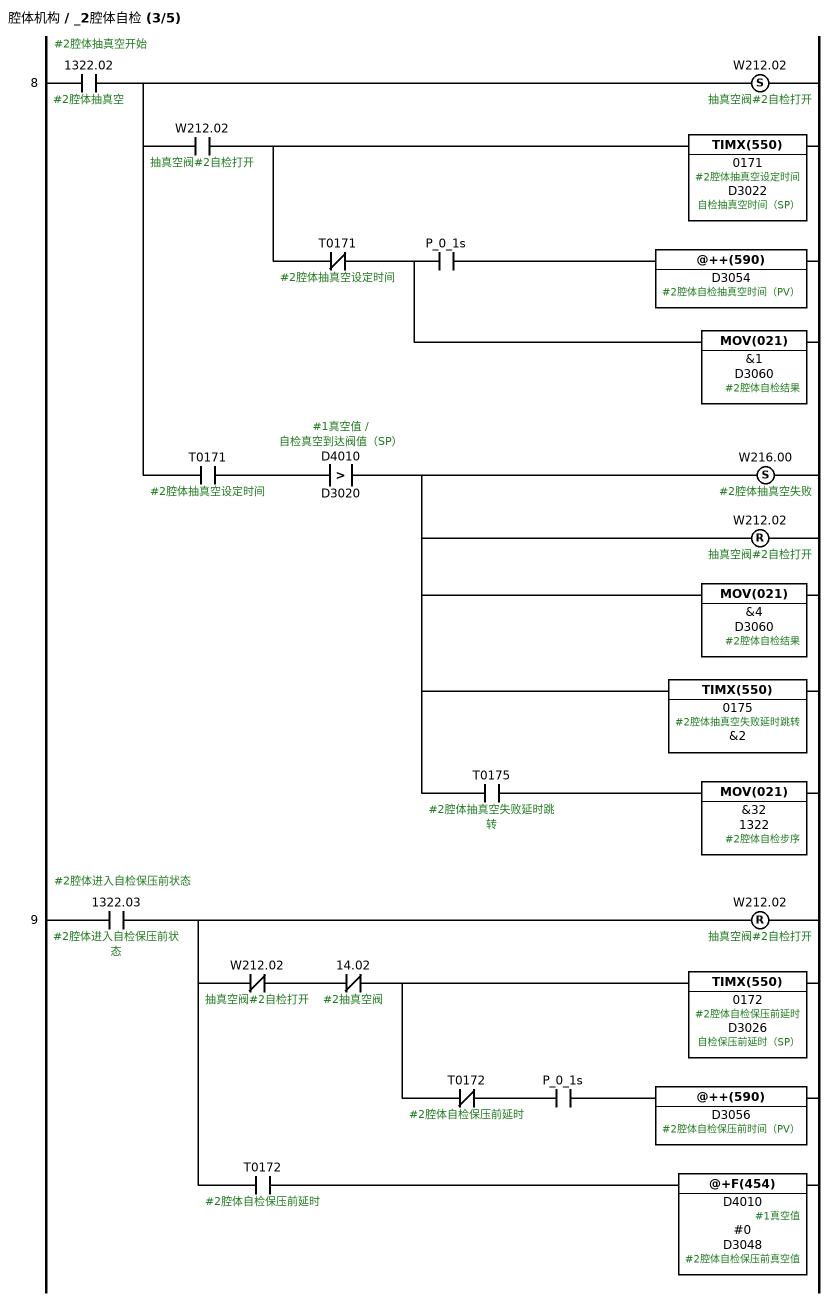
; [picture p312: 腔体机构 / _2腔体自检, rungs 8-9]
; rung 8: #2腔体抽真空开始
LD 1322.02  ; #2腔体抽真空
OUT TR0
SET W212.02  ; 抽真空阀#2自检打开
AND W212.02  ; 抽真空阀#2自检打开
TIMX(550) 0171 D3022  ; 自检抽真空时间（SP）, #2腔体抽真空设定时间
ANDNOT T0171  ; #2腔体抽真空设定时间
OUT TR1
AND P_0_1s
@++(590) D3054  ; #2腔体自检抽真空时间（PV）
LD TR1
MOV(021) &1 D3060  ; #2腔体自检结果
LD TR0
AND T0171  ; #2腔体抽真空设定时间
AND>F(333) D4010 D3020  ; #1真空值, 自检真空到达阀值（SP）
SET W216.00  ; #2腔体抽真空失败
RSET W212.02  ; 抽真空阀#2自检打开
MOV(021) &4 D3060  ; #2腔体自检结果
TIMX(550) 0175 &2  ; #2腔体抽真空失败延时跳转
AND T0175  ; #2腔体抽真空失败延时跳转
MOV(021) &32 1322  ; #2腔体自检步序
; rung 9: #2腔体进入自检保压前状态
LD 1322.03  ; #2腔体进入自检保压前状态
OUT TR0
RSET W212.02  ; 抽真空阀#2自检打开
ANDNOT W212.02  ; 抽真空阀#2自检打开
ANDNOT 14.02  ; #2抽真空阀
TIMX(550) 0172 D3026  ; 自检保压前延时（SP）, #2腔体自检保压前延时
ANDNOT T0172  ; #2腔体自检保压前延时
AND P_0_1s
@++(590) D3056  ; #2腔体自检保压前时间（PV）
LD TR0
AND T0172  ; #2腔体自检保压前延时
@+F(454) D4010 #0 D3048  ; #1真空值, #2腔体自检保压前真空值

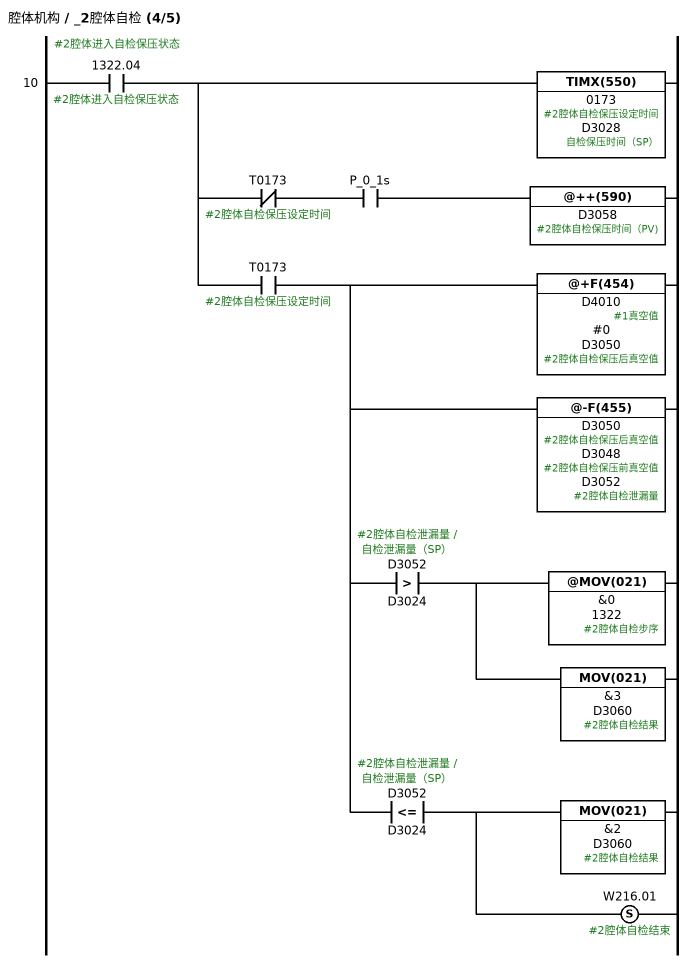
; rung 10: #2腔体进入自检保压状态
LD 1322.04  ; #2腔体进入自检保压状态
OUT TR0
TIMX(550) 0173 D3028  ; 自检保压时间（SP）, #2腔体自检保压设定时间
ANDNOT T0173  ; #2腔体自检保压设定时间
AND P_0_1s
@++(590) D3058  ; #2腔体自检保压时间（PV)
LD TR0
AND T0173  ; #2腔体自检保压设定时间
OUT TR0
@+F(454) D4010 #0 D3050  ; #1真空值, #2腔体自检保压后真空值
@-F(455) D3050 D3048 D3052  ; #2腔体自检保压后真空值, #2腔体自检保压前真空值, #2腔体自检泄漏量
AND>F(333) D3052 D3024  ; #2腔体自检泄漏量, 自检泄漏量（SP）
@MOV(021) &0 1322  ; #2腔体自检步序
MOV(021) &3 D3060  ; #2腔体自检结果
LD TR0
AND<=F(332) D3052 D3024  ; #2腔体自检泄漏量, 自检泄漏量（SP）
MOV(021) &2 D3060  ; #2腔体自检结果
SET W216.01  ; #2腔体自检结束

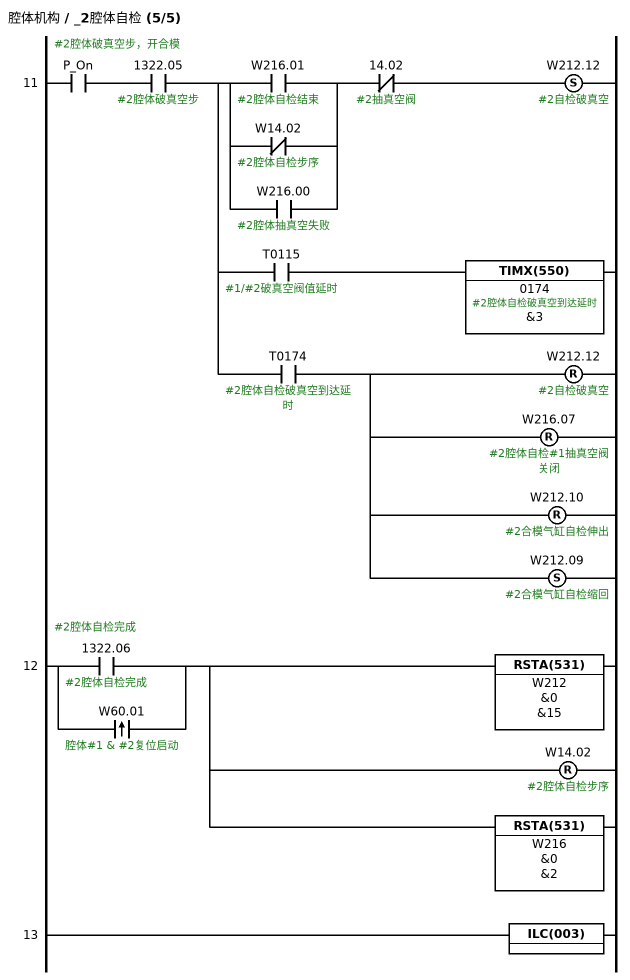
; rung 11: #2腔体破真空步，开合模
LD P_On
AND 1322.05  ; #2腔体破真空步
OUT TR0
LD W216.01  ; #2腔体自检结束
ORNOT W14.02  ; #2腔体自检步序
OR W216.00  ; #2腔体抽真空失败
ANDLD
ANDNOT 14.02  ; #2抽真空阀
SET W212.12  ; #2自检破真空
LD TR0
AND T0115  ; #1/#2破真空阀值延时
TIMX(550) 0174 &3  ; #2腔体自检破真空到达延时
LD TR0
AND T0174  ; #2腔体自检破真空到达延时
RSET W212.12  ; #2自检破真空
RSET W216.07  ; #2腔体自检#1抽真空阀关闭
RSET W212.10  ; #2合模气缸自检伸出
SET W212.09  ; #2合模气缸自检缩回
; rung 12: #2腔体自检完成
LD 1322.06  ; #2腔体自检完成
@OR W60.01  ; 腔体#1 & #2复位启动
RSTA(531) W212 &0 &15
RSET W14.02  ; #2腔体自检步序
RSTA(531) W216 &0 &2
; rung 13
ILC(003)

### Section _3腔体自检

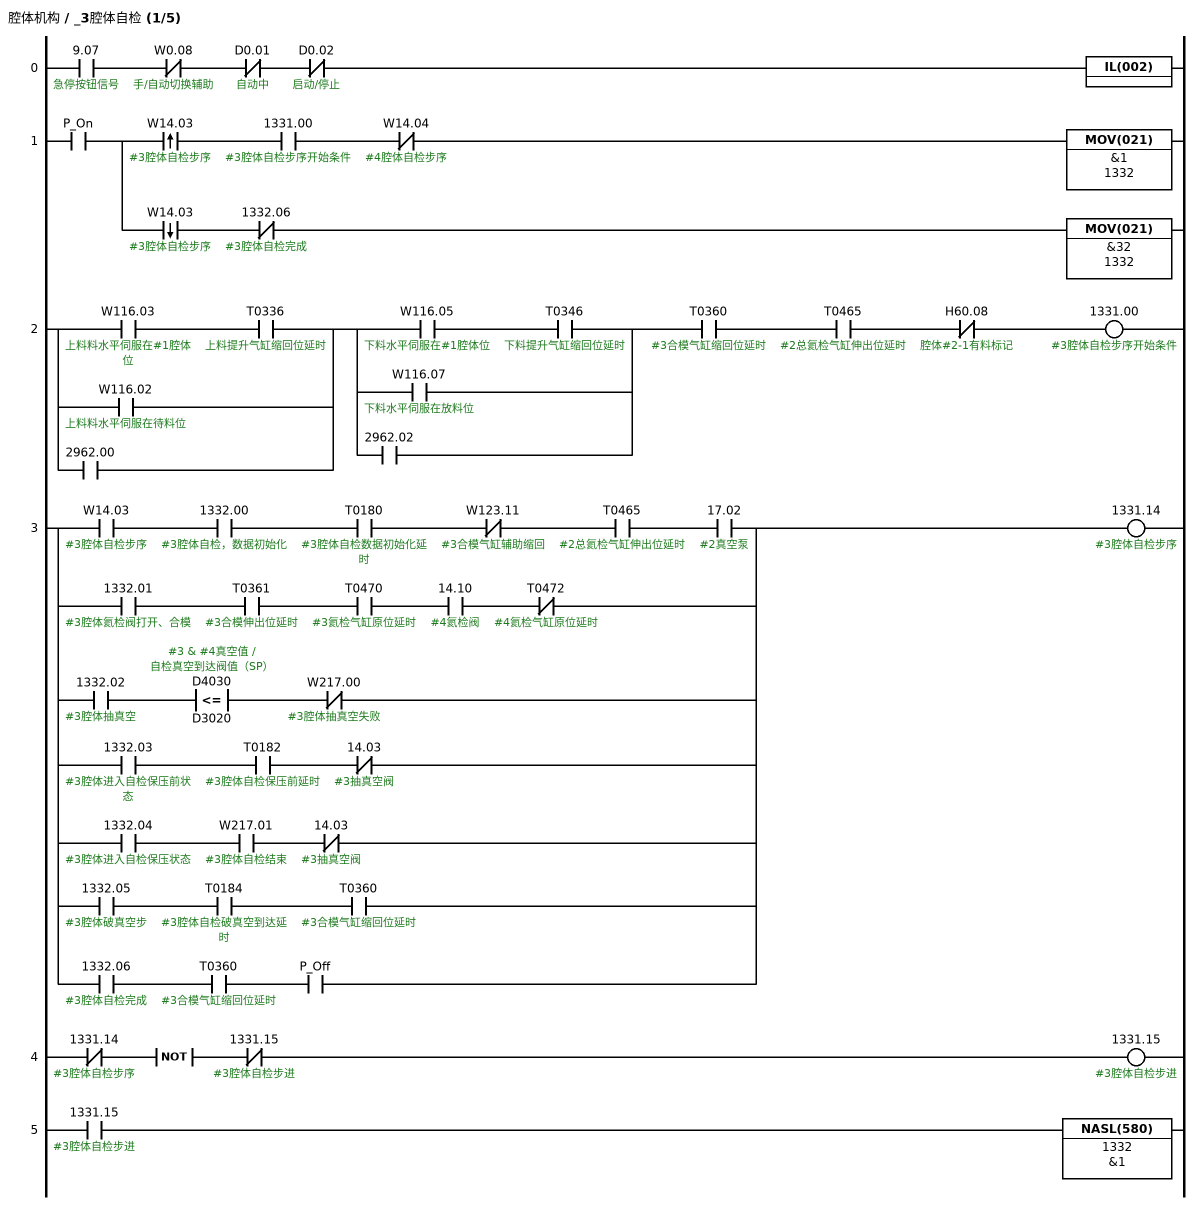
; rung 0
LD 9.07  ; 急停按钮信号
ANDNOT W0.08  ; 手/自动切换辅助
ANDNOT D0.01  ; 自动中
ANDNOT D0.02  ; 启动/停止
IL(002)
; rung 1
LD P_On
OUT TR0
@AND W14.03  ; #3腔体自检步序
AND 1331.00  ; #3腔体自检步序开始条件
ANDNOT W14.04  ; #4腔体自检步序
MOV(021) &1 1332
LD TR0
%AND W14.03  ; #3腔体自检步序
ANDNOT 1332.06  ; #3腔体自检完成
MOV(021) &32 1332
; rung 2
LD W116.03  ; 上料料水平伺服在#1腔体位
AND T0336  ; 上料提升气缸缩回位延时
OR W116.02  ; 上料料水平伺服在待料位
OR 2962.00
LD W116.05  ; 下料水平伺服在#1腔体位
AND T0346  ; 下料提升气缸缩回位延时
OR W116.07  ; 下料水平伺服在放料位
OR 2962.02
ANDLD
AND T0360  ; #3合模气缸缩回位延时
AND T0465  ; #2总氦检气缸伸出位延时
ANDNOT H60.08  ; 腔体#2-1有料标记
OUT 1331.00  ; #3腔体自检步序开始条件
; rung 3
LD W14.03  ; #3腔体自检步序
AND 1332.00  ; #3腔体自检，数据初始化
AND T0180  ; #3腔体自检数据初始化延时
ANDNOT W123.11  ; #3合模气缸辅助缩回
AND T0465  ; #2总氦检气缸伸出位延时
AND 17.02  ; #2真空泵
LD 1332.01  ; #3腔体氦检阀打开、合模
AND T0361  ; #3合模伸出位延时
AND T0470  ; #3氦检气缸原位延时
AND 14.10  ; #4氦检阀
ANDNOT T0472  ; #4氦检气缸原位延时
ORLD
LD 1332.02  ; #3腔体抽真空
AND<=F(332) D4030 D3020  ; #3 & #4真空值, 自检真空到达阀值（SP）
ANDNOT W217.00  ; #3腔体抽真空失败
ORLD
LD 1332.03  ; #3腔体进入自检保压前状态
AND T0182  ; #3腔体自检保压前延时
ANDNOT 14.03  ; #3抽真空阀
ORLD
LD 1332.04  ; #3腔体进入自检保压状态
AND W217.01  ; #3腔体自检结束
ANDNOT 14.03  ; #3抽真空阀
ORLD
LD 1332.05  ; #3腔体破真空步
AND T0184  ; #3腔体自检破真空到达延时
AND T0360  ; #3合模气缸缩回位延时
ORLD
LD 1332.06  ; #3腔体自检完成
AND T0360  ; #3合模气缸缩回位延时
AND P_Off
ORLD
OUT 1331.14  ; #3腔体自检步序
; rung 4
LDNOT 1331.14  ; #3腔体自检步序
NOT(520)
ANDNOT 1331.15  ; #3腔体自检步进
OUT 1331.15  ; #3腔体自检步进
; rung 5
LD 1331.15  ; #3腔体自检步进
NASL(580) 1332 &1

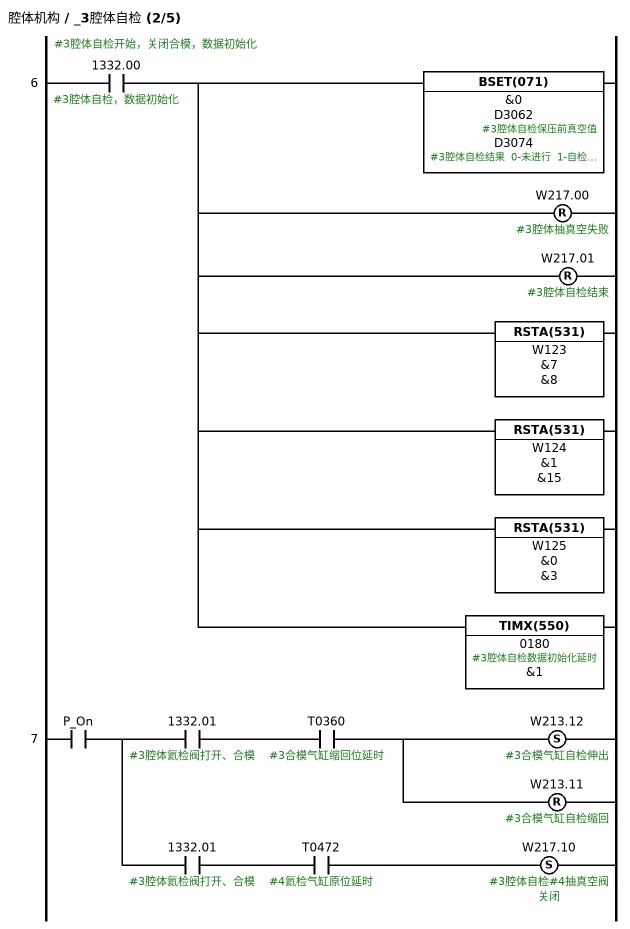
; rung 6: #3腔体自检开始，关闭合模，数据初始化
LD 1332.00  ; #3腔体自检，数据初始化
BSET(071) &0 D3062 D3074  ; #3腔体自检保压前真空值, #3腔体自检结果  0-未进行  1-自检中  2-自检OK  3-自检泄漏  4-自检抽真空NG
RSET W217.00  ; #3腔体抽真空失败
RSET W217.01  ; #3腔体自检结束
RSTA(531) W123 &7 &8
RSTA(531) W124 &1 &15
RSTA(531) W125 &0 &3
TIMX(550) 0180 &1  ; #3腔体自检数据初始化延时
; rung 7
LD P_On
OUT TR0
AND 1332.01  ; #3腔体氦检阀打开、合模
AND T0360  ; #3合模气缸缩回位延时
SET W213.12  ; #3合模气缸自检伸出
RSET W213.11  ; #3合模气缸自检缩回
LD TR0
AND 1332.01  ; #3腔体氦检阀打开、合模
AND T0472  ; #4氦检气缸原位延时
SET W217.10  ; #3腔体自检#4抽真空阀关闭

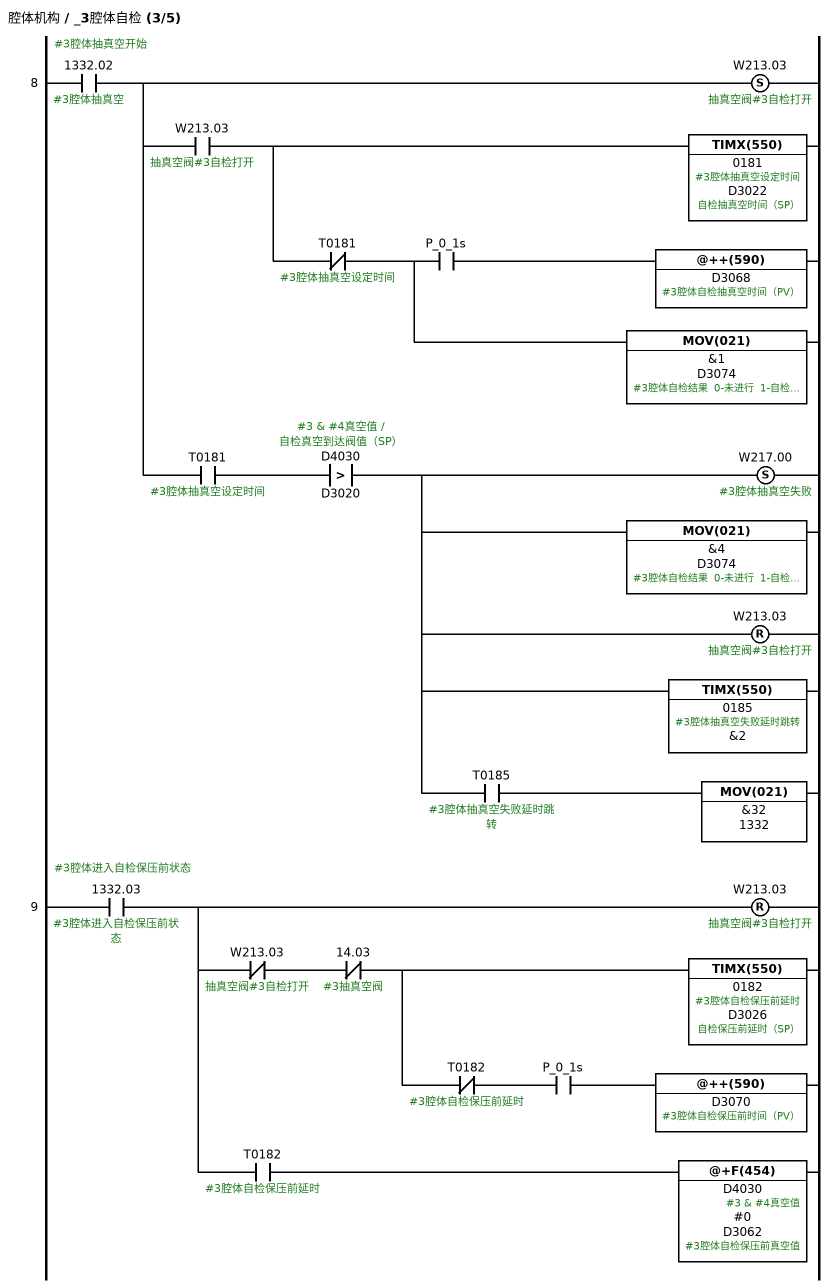
; rung 8: #3腔体抽真空开始
LD 1332.02  ; #3腔体抽真空
OUT TR0
SET W213.03  ; 抽真空阀#3自检打开
AND W213.03  ; 抽真空阀#3自检打开
TIMX(550) 0181 D3022  ; 自检抽真空时间（SP）, #3腔体抽真空设定时间
ANDNOT T0181  ; #3腔体抽真空设定时间
OUT TR1
AND P_0_1s
@++(590) D3068  ; #3腔体自检抽真空时间（PV）
LD TR1
MOV(021) &1 D3074  ; #3腔体自检结果  0-未进行  1-自检中  2-自检OK  3-自检泄漏  4-自检抽真空NG
LD TR0
AND T0181  ; #3腔体抽真空设定时间
AND>F(333) D4030 D3020  ; #3 & #4真空值, 自检真空到达阀值（SP）
SET W217.00  ; #3腔体抽真空失败
MOV(021) &4 D3074  ; #3腔体自检结果  0-未进行  1-自检中  2-自检OK  3-自检泄漏  4-自检抽真空NG
RSET W213.03  ; 抽真空阀#3自检打开
TIMX(550) 0185 &2  ; #3腔体抽真空失败延时跳转
AND T0185  ; #3腔体抽真空失败延时跳转
MOV(021) &32 1332
; rung 9: #3腔体进入自检保压前状态
LD 1332.03  ; #3腔体进入自检保压前状态
OUT TR0
RSET W213.03  ; 抽真空阀#3自检打开
ANDNOT W213.03  ; 抽真空阀#3自检打开
ANDNOT 14.03  ; #3抽真空阀
TIMX(550) 0182 D3026  ; 自检保压前延时（SP）, #3腔体自检保压前延时
ANDNOT T0182  ; #3腔体自检保压前延时
AND P_0_1s
@++(590) D3070  ; #3腔体自检保压前时间（PV）
LD TR0
AND T0182  ; #3腔体自检保压前延时
@+F(454) D4030 #0 D3062  ; #3 & #4真空值, #3腔体自检保压前真空值

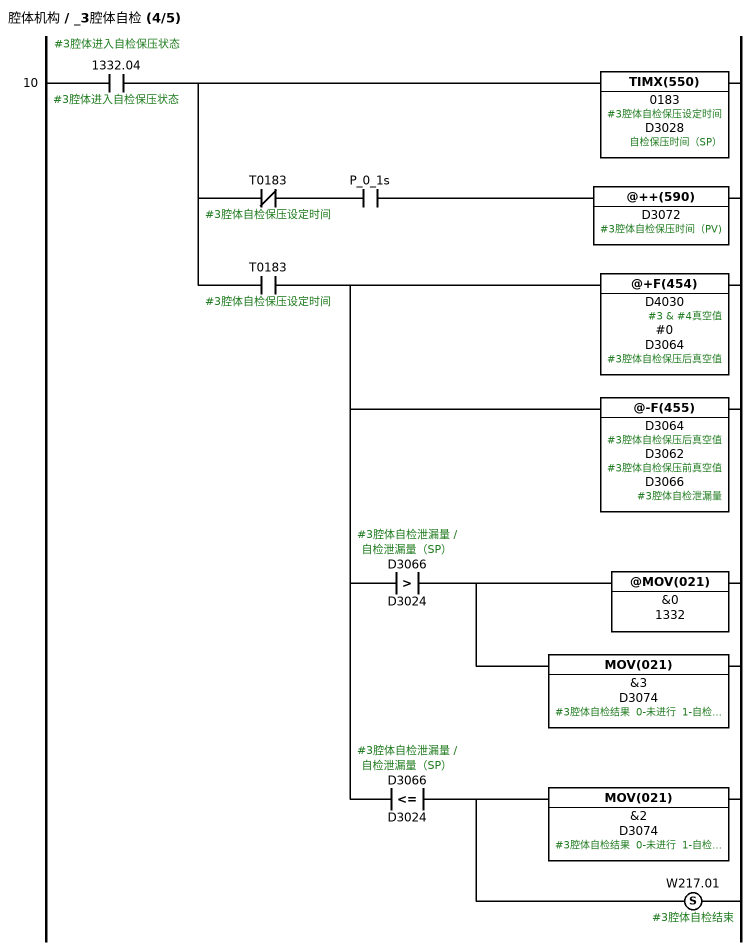
; rung 10: #3腔体进入自检保压状态
LD 1332.04  ; #3腔体进入自检保压状态
OUT TR0
TIMX(550) 0183 D3028  ; 自检保压时间（SP）, #3腔体自检保压设定时间
ANDNOT T0183  ; #3腔体自检保压设定时间
AND P_0_1s
@++(590) D3072  ; #3腔体自检保压时间（PV)
LD TR0
AND T0183  ; #3腔体自检保压设定时间
OUT TR0
@+F(454) D4030 #0 D3064  ; #3 & #4真空值, #3腔体自检保压后真空值
@-F(455) D3064 D3062 D3066  ; #3腔体自检保压后真空值, #3腔体自检保压前真空值, #3腔体自检泄漏量
AND>F(333) D3066 D3024  ; #3腔体自检泄漏量, 自检泄漏量（SP）
@MOV(021) &0 1332
MOV(021) &3 D3074  ; #3腔体自检结果  0-未进行  1-自检中  2-自检OK  3-自检泄漏  4-自检抽真空NG
LD TR0
AND<=F(332) D3066 D3024  ; #3腔体自检泄漏量, 自检泄漏量（SP）
MOV(021) &2 D3074  ; #3腔体自检结果  0-未进行  1-自检中  2-自检OK  3-自检泄漏  4-自检抽真空NG
SET W217.01  ; #3腔体自检结束

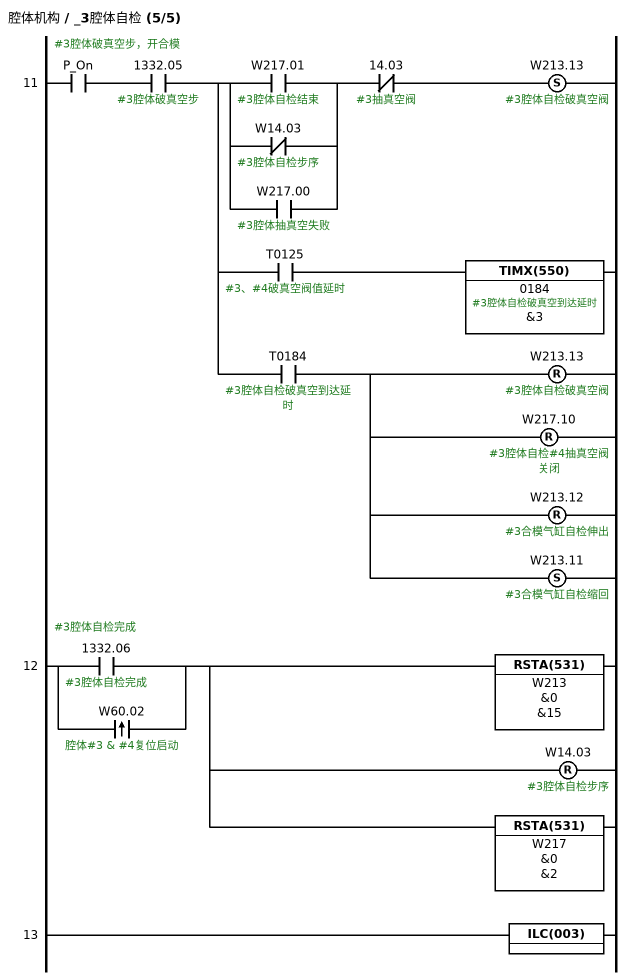
; rung 11: #3腔体破真空步，开合模
LD P_On
AND 1332.05  ; #3腔体破真空步
OUT TR0
LD W217.01  ; #3腔体自检结束
ORNOT W14.03  ; #3腔体自检步序
OR W217.00  ; #3腔体抽真空失败
ANDLD
ANDNOT 14.03  ; #3抽真空阀
SET W213.13  ; #3腔体自检破真空阀
LD TR0
AND T0125  ; #3、#4破真空阀值延时
TIMX(550) 0184 &3  ; #3腔体自检破真空到达延时
LD TR0
AND T0184  ; #3腔体自检破真空到达延时
RSET W213.13  ; #3腔体自检破真空阀
RSET W217.10  ; #3腔体自检#4抽真空阀关闭
RSET W213.12  ; #3合模气缸自检伸出
SET W213.11  ; #3合模气缸自检缩回
; rung 12: #3腔体自检完成
LD 1332.06  ; #3腔体自检完成
@OR W60.02  ; 腔体#3 & #4复位启动
RSTA(531) W213 &0 &15
RSET W14.03  ; #3腔体自检步序
RSTA(531) W217 &0 &2
; rung 13
ILC(003)

### Section _4腔体自检

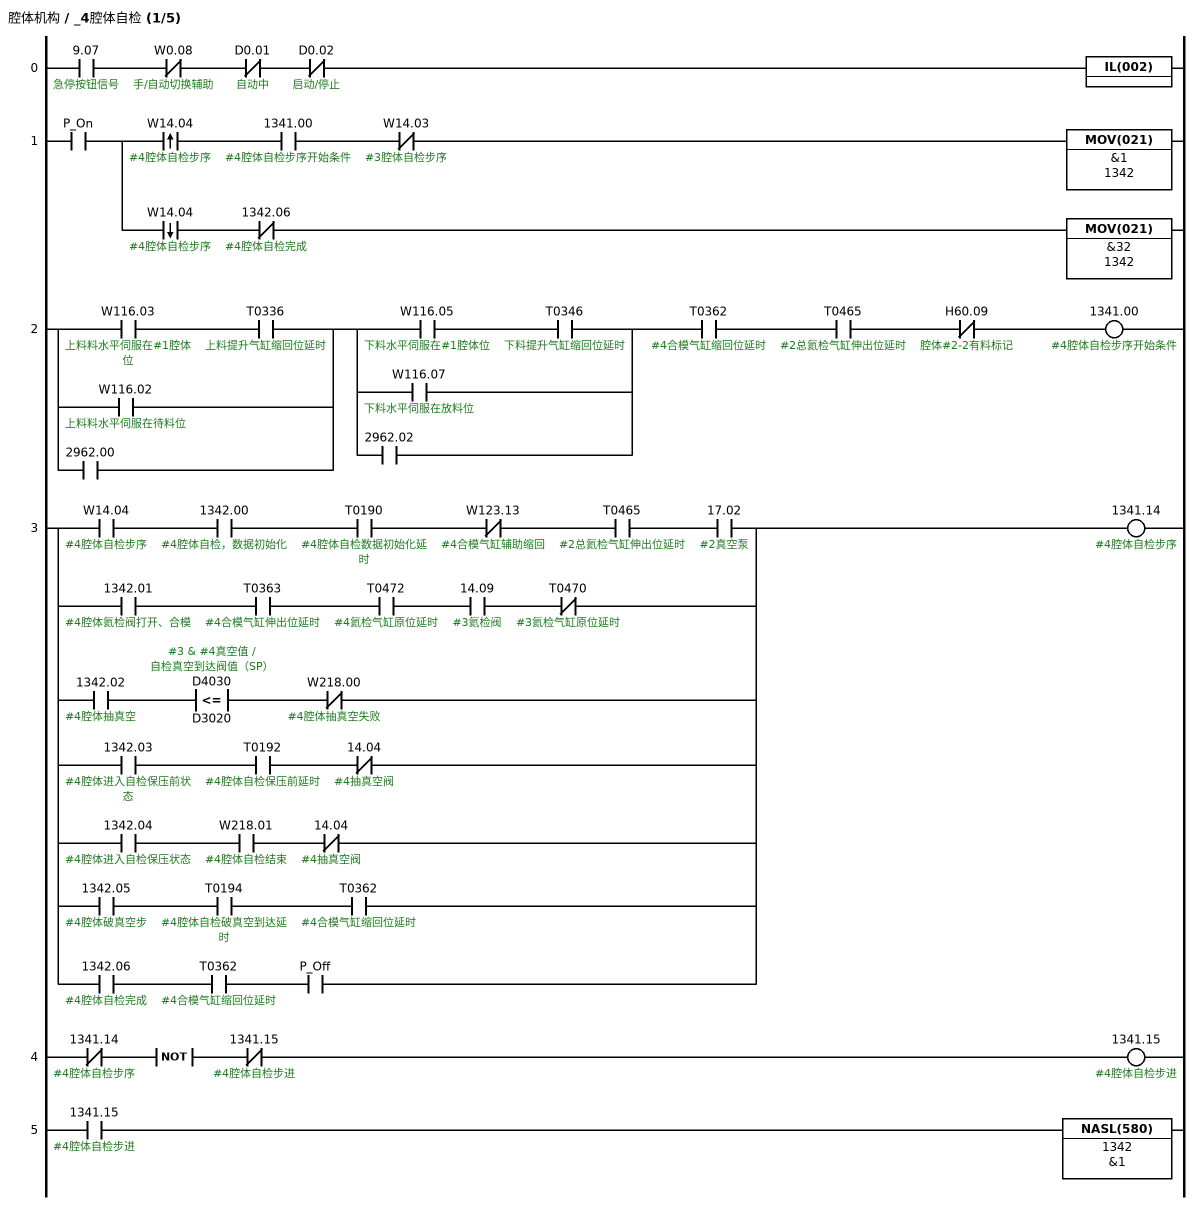
; rung 0
LD 9.07  ; 急停按钮信号
ANDNOT W0.08  ; 手/自动切换辅助
ANDNOT D0.01  ; 自动中
ANDNOT D0.02  ; 启动/停止
IL(002)
; rung 1
LD P_On
OUT TR0
@AND W14.04  ; #4腔体自检步序
AND 1341.00  ; #4腔体自检步序开始条件
ANDNOT W14.03  ; #3腔体自检步序
MOV(021) &1 1342
LD TR0
%AND W14.04  ; #4腔体自检步序
ANDNOT 1342.06  ; #4腔体自检完成
MOV(021) &32 1342
; rung 2
LD W116.03  ; 上料料水平伺服在#1腔体位
AND T0336  ; 上料提升气缸缩回位延时
OR W116.02  ; 上料料水平伺服在待料位
OR 2962.00
LD W116.05  ; 下料水平伺服在#1腔体位
AND T0346  ; 下料提升气缸缩回位延时
OR W116.07  ; 下料水平伺服在放料位
OR 2962.02
ANDLD
AND T0362  ; #4合模气缸缩回位延时
AND T0465  ; #2总氦检气缸伸出位延时
ANDNOT H60.09  ; 腔体#2-2有料标记
OUT 1341.00  ; #4腔体自检步序开始条件
; rung 3
LD W14.04  ; #4腔体自检步序
AND 1342.00  ; #4腔体自检，数据初始化
AND T0190  ; #4腔体自检数据初始化延时
ANDNOT W123.13  ; #4合模气缸辅助缩回
AND T0465  ; #2总氦检气缸伸出位延时
AND 17.02  ; #2真空泵
LD 1342.01  ; #4腔体氦检阀打开、合模
AND T0363  ; #4合模气缸伸出位延时
AND T0472  ; #4氦检气缸原位延时
AND 14.09  ; #3氦检阀
ANDNOT T0470  ; #3氦检气缸原位延时
ORLD
LD 1342.02  ; #4腔体抽真空
AND<=F(332) D4030 D3020  ; #3 & #4真空值, 自检真空到达阀值（SP）
ANDNOT W218.00  ; #4腔体抽真空失败
ORLD
LD 1342.03  ; #4腔体进入自检保压前状态
AND T0192  ; #4腔体自检保压前延时
ANDNOT 14.04  ; #4抽真空阀
ORLD
LD 1342.04  ; #4腔体进入自检保压状态
AND W218.01  ; #4腔体自检结束
ANDNOT 14.04  ; #4抽真空阀
ORLD
LD 1342.05  ; #4腔体破真空步
AND T0194  ; #4腔体自检破真空到达延时
AND T0362  ; #4合模气缸缩回位延时
ORLD
LD 1342.06  ; #4腔体自检完成
AND T0362  ; #4合模气缸缩回位延时
AND P_Off
ORLD
OUT 1341.14  ; #4腔体自检步序
; rung 4
LDNOT 1341.14  ; #4腔体自检步序
NOT(520)
ANDNOT 1341.15  ; #4腔体自检步进
OUT 1341.15  ; #4腔体自检步进
; rung 5
LD 1341.15  ; #4腔体自检步进
NASL(580) 1342 &1

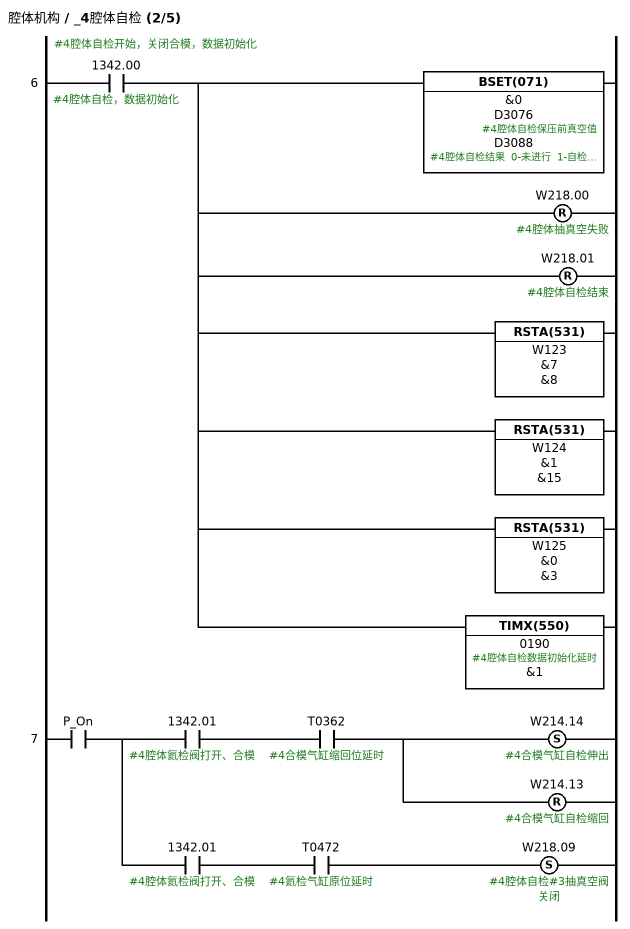
; rung 6: #4腔体自检开始，关闭合模，数据初始化
LD 1342.00  ; #4腔体自检，数据初始化
BSET(071) &0 D3076 D3088  ; #4腔体自检保压前真空值, #4腔体自检结果  0-未进行  1-自检中  2-自检OK  3-自检泄漏  4-自检抽真空NG
RSET W218.00  ; #4腔体抽真空失败
RSET W218.01  ; #4腔体自检结束
RSTA(531) W123 &7 &8
RSTA(531) W124 &1 &15
RSTA(531) W125 &0 &3
TIMX(550) 0190 &1  ; #4腔体自检数据初始化延时
; rung 7
LD P_On
OUT TR0
AND 1342.01  ; #4腔体氦检阀打开、合模
AND T0362  ; #4合模气缸缩回位延时
SET W214.14  ; #4合模气缸自检伸出
RSET W214.13  ; #4合模气缸自检缩回
LD TR0
AND 1342.01  ; #4腔体氦检阀打开、合模
AND T0472  ; #4氦检气缸原位延时
SET W218.09  ; #4腔体自检#3抽真空阀关闭

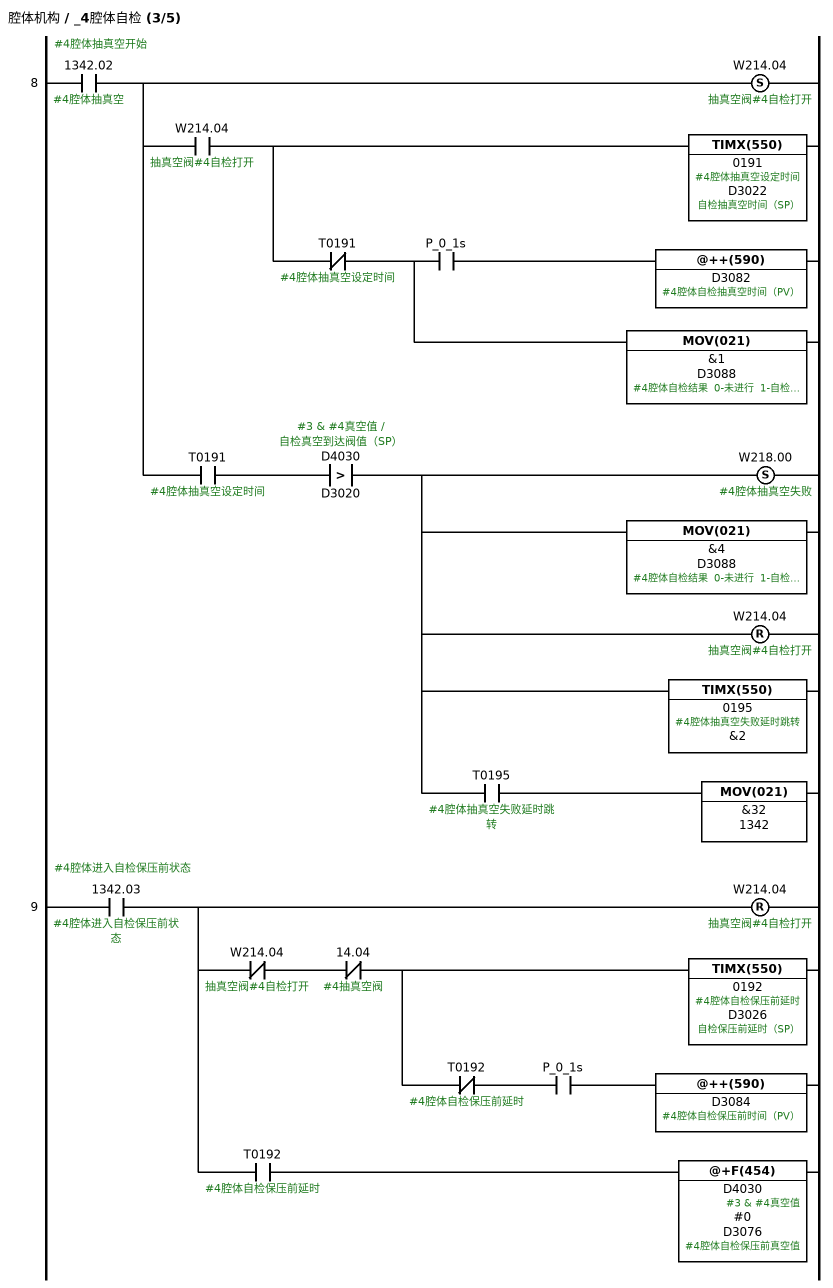
; rung 8: #4腔体抽真空开始
LD 1342.02  ; #4腔体抽真空
OUT TR0
SET W214.04  ; 抽真空阀#4自检打开
AND W214.04  ; 抽真空阀#4自检打开
TIMX(550) 0191 D3022  ; 自检抽真空时间（SP）, #4腔体抽真空设定时间
ANDNOT T0191  ; #4腔体抽真空设定时间
OUT TR1
AND P_0_1s
@++(590) D3082  ; #4腔体自检抽真空时间（PV）
LD TR1
MOV(021) &1 D3088  ; #4腔体自检结果  0-未进行  1-自检中  2-自检OK  3-自检泄漏  4-自检抽真空NG
LD TR0
AND T0191  ; #4腔体抽真空设定时间
AND>F(333) D4030 D3020  ; #3 & #4真空值, 自检真空到达阀值（SP）
SET W218.00  ; #4腔体抽真空失败
MOV(021) &4 D3088  ; #4腔体自检结果  0-未进行  1-自检中  2-自检OK  3-自检泄漏  4-自检抽真空NG
RSET W214.04  ; 抽真空阀#4自检打开
TIMX(550) 0195 &2  ; #4腔体抽真空失败延时跳转
AND T0195  ; #4腔体抽真空失败延时跳转
MOV(021) &32 1342
; rung 9: #4腔体进入自检保压前状态
LD 1342.03  ; #4腔体进入自检保压前状态
OUT TR0
RSET W214.04  ; 抽真空阀#4自检打开
ANDNOT W214.04  ; 抽真空阀#4自检打开
ANDNOT 14.04  ; #4抽真空阀
TIMX(550) 0192 D3026  ; 自检保压前延时（SP）, #4腔体自检保压前延时
ANDNOT T0192  ; #4腔体自检保压前延时
AND P_0_1s
@++(590) D3084  ; #4腔体自检保压前时间（PV）
LD TR0
AND T0192  ; #4腔体自检保压前延时
@+F(454) D4030 #0 D3076  ; #3 & #4真空值, #4腔体自检保压前真空值

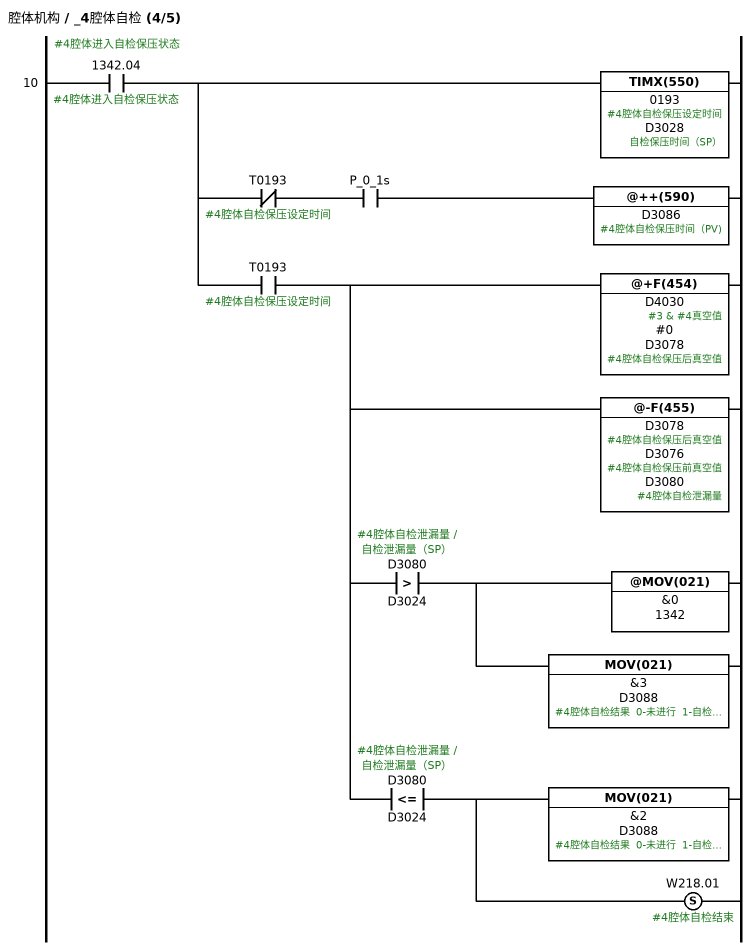
; rung 10: #4腔体进入自检保压状态
LD 1342.04  ; #4腔体进入自检保压状态
OUT TR0
TIMX(550) 0193 D3028  ; 自检保压时间（SP）, #4腔体自检保压设定时间
ANDNOT T0193  ; #4腔体自检保压设定时间
AND P_0_1s
@++(590) D3086  ; #4腔体自检保压时间（PV)
LD TR0
AND T0193  ; #4腔体自检保压设定时间
OUT TR0
@+F(454) D4030 #0 D3078  ; #3 & #4真空值, #4腔体自检保压后真空值
@-F(455) D3078 D3076 D3080  ; #4腔体自检保压后真空值, #4腔体自检保压前真空值, #4腔体自检泄漏量
AND>F(333) D3080 D3024  ; #4腔体自检泄漏量, 自检泄漏量（SP）
@MOV(021) &0 1342
MOV(021) &3 D3088  ; #4腔体自检结果  0-未进行  1-自检中  2-自检OK  3-自检泄漏  4-自检抽真空NG
LD TR0
AND<=F(332) D3080 D3024  ; #4腔体自检泄漏量, 自检泄漏量（SP）
MOV(021) &2 D3088  ; #4腔体自检结果  0-未进行  1-自检中  2-自检OK  3-自检泄漏  4-自检抽真空NG
SET W218.01  ; #4腔体自检结束

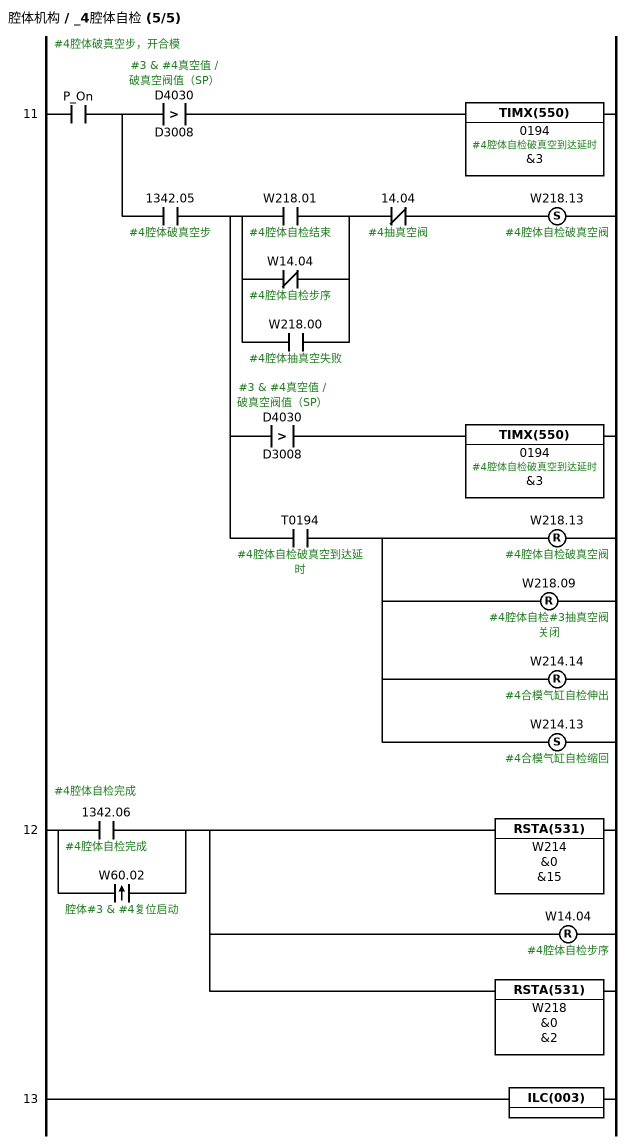
; rung 11: #4腔体破真空步，开合模
LD P_On
OUT TR0
AND>F(333) D4030 D3008  ; #3 & #4真空值, 破真空阀值（SP）
TIMX(550) 0194 &3  ; #4腔体自检破真空到达延时
LD TR0
AND 1342.05  ; #4腔体破真空步
OUT TR0
LD W218.01  ; #4腔体自检结束
ORNOT W14.04  ; #4腔体自检步序
OR W218.00  ; #4腔体抽真空失败
ANDLD
ANDNOT 14.04  ; #4抽真空阀
SET W218.13  ; #4腔体自检破真空阀
LD TR0
AND>F(333) D4030 D3008  ; #3 & #4真空值, 破真空阀值（SP）
TIMX(550) 0194 &3  ; #4腔体自检破真空到达延时
LD TR0
AND T0194  ; #4腔体自检破真空到达延时
RSET W218.13  ; #4腔体自检破真空阀
RSET W218.09  ; #4腔体自检#3抽真空阀关闭
RSET W214.14  ; #4合模气缸自检伸出
SET W214.13  ; #4合模气缸自检缩回
; rung 12: #4腔体自检完成
LD 1342.06  ; #4腔体自检完成
@OR W60.02  ; 腔体#3 & #4复位启动
RSTA(531) W214 &0 &15
RSET W14.04  ; #4腔体自检步序
RSTA(531) W218 &0 &2
; rung 13
ILC(003)

### Section 腔体机构输出

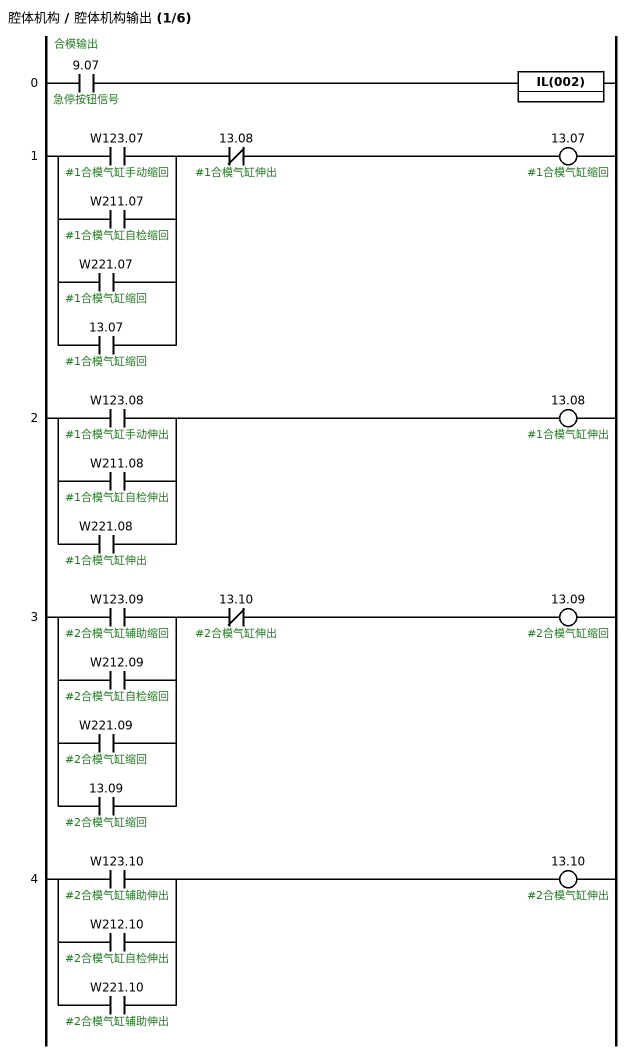
; rung 0: 合模输出
LD 9.07  ; 急停按钮信号
IL(002)
; rung 1
LD W123.07  ; #1合模气缸手动缩回
OR W211.07  ; #1合模气缸自检缩回
OR W221.07  ; #1合模气缸缩回
OR 13.07  ; #1合模气缸缩回
ANDNOT 13.08  ; #1合模气缸伸出
OUT 13.07  ; #1合模气缸缩回
; rung 2
LD W123.08  ; #1合模气缸手动伸出
OR W211.08  ; #1合模气缸自检伸出
OR W221.08  ; #1合模气缸伸出
OUT 13.08  ; #1合模气缸伸出
; rung 3
LD W123.09  ; #2合模气缸辅助缩回
OR W212.09  ; #2合模气缸自检缩回
OR W221.09  ; #2合模气缸缩回
OR 13.09  ; #2合模气缸缩回
ANDNOT 13.10  ; #2合模气缸伸出
OUT 13.09  ; #2合模气缸缩回
; rung 4
LD W123.10  ; #2合模气缸辅助伸出
OR W212.10  ; #2合模气缸自检伸出
OR W221.10  ; #2合模气缸辅助伸出
OUT 13.10  ; #2合模气缸伸出

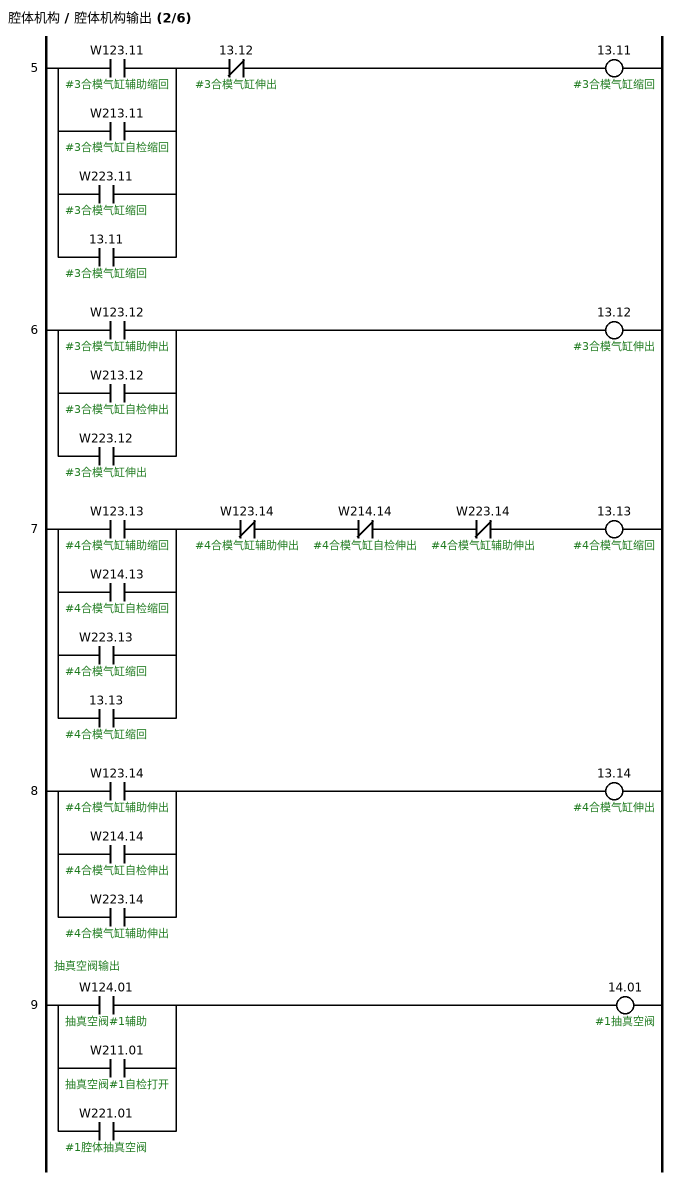
; rung 5
LD W123.11  ; #3合模气缸辅助缩回
OR W213.11  ; #3合模气缸自检缩回
OR W223.11  ; #3合模气缸缩回
OR 13.11  ; #3合模气缸缩回
ANDNOT 13.12  ; #3合模气缸伸出
OUT 13.11  ; #3合模气缸缩回
; rung 6
LD W123.12  ; #3合模气缸辅助伸出
OR W213.12  ; #3合模气缸自检伸出
OR W223.12  ; #3合模气缸伸出
OUT 13.12  ; #3合模气缸伸出
; rung 7
LD W123.13  ; #4合模气缸辅助缩回
OR W214.13  ; #4合模气缸自检缩回
OR W223.13  ; #4合模气缸缩回
OR 13.13  ; #4合模气缸缩回
ANDNOT W123.14  ; #4合模气缸辅助伸出
ANDNOT W214.14  ; #4合模气缸自检伸出
ANDNOT W223.14  ; #4合模气缸辅助伸出
OUT 13.13  ; #4合模气缸缩回
; rung 8
LD W123.14  ; #4合模气缸辅助伸出
OR W214.14  ; #4合模气缸自检伸出
OR W223.14  ; #4合模气缸辅助伸出
OUT 13.14  ; #4合模气缸伸出
; rung 9: 抽真空阀输出
LD W124.01  ; 抽真空阀#1辅助
OR W211.01  ; 抽真空阀#1自检打开
OR W221.01  ; #1腔体抽真空阀
OUT 14.01  ; #1抽真空阀

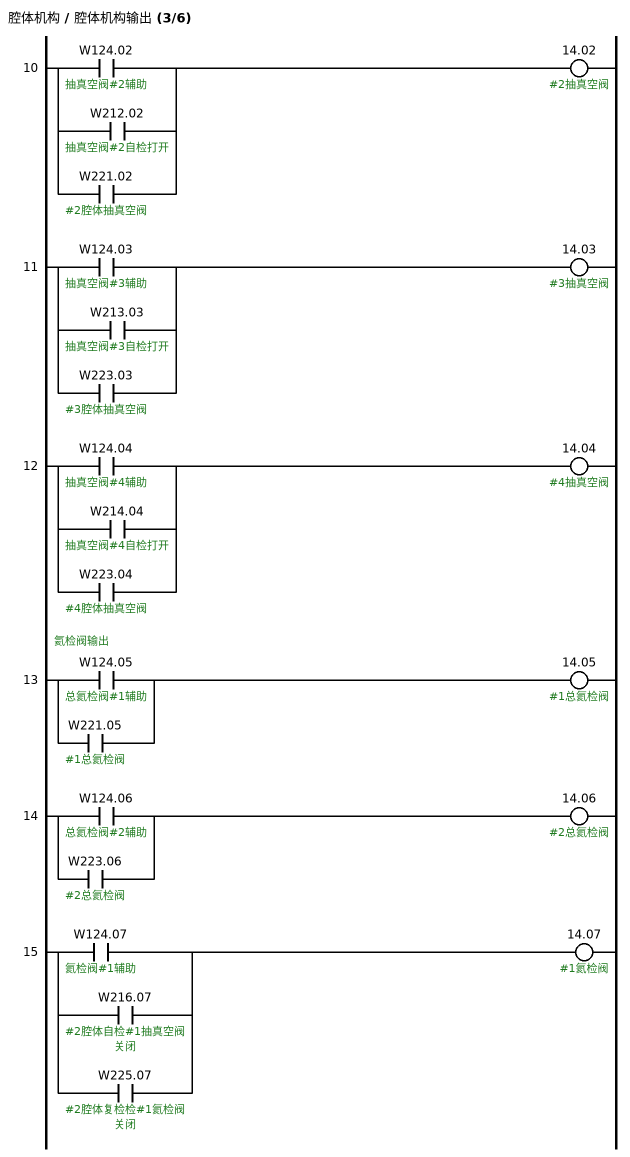
; rung 10
LD W124.02  ; 抽真空阀#2辅助
OR W212.02  ; 抽真空阀#2自检打开
OR W221.02  ; #2腔体抽真空阀
OUT 14.02  ; #2抽真空阀
; rung 11
LD W124.03  ; 抽真空阀#3辅助
OR W213.03  ; 抽真空阀#3自检打开
OR W223.03  ; #3腔体抽真空阀
OUT 14.03  ; #3抽真空阀
; rung 12
LD W124.04  ; 抽真空阀#4辅助
OR W214.04  ; 抽真空阀#4自检打开
OR W223.04  ; #4腔体抽真空阀
OUT 14.04  ; #4抽真空阀
; rung 13: 氦检阀输出
LD W124.05  ; 总氦检阀#1辅助
OR W221.05  ; #1总氦检阀
OUT 14.05  ; #1总氦检阀
; rung 14
LD W124.06  ; 总氦检阀#2辅助
OR W223.06  ; #2总氦检阀
OUT 14.06  ; #2总氦检阀
; rung 15
LD W124.07  ; 氦检阀#1辅助
OR W216.07  ; #2腔体自检#1抽真空阀关闭
OR W225.07  ; #2腔体复检检#1氦检阀关闭
OUT 14.07  ; #1氦检阀

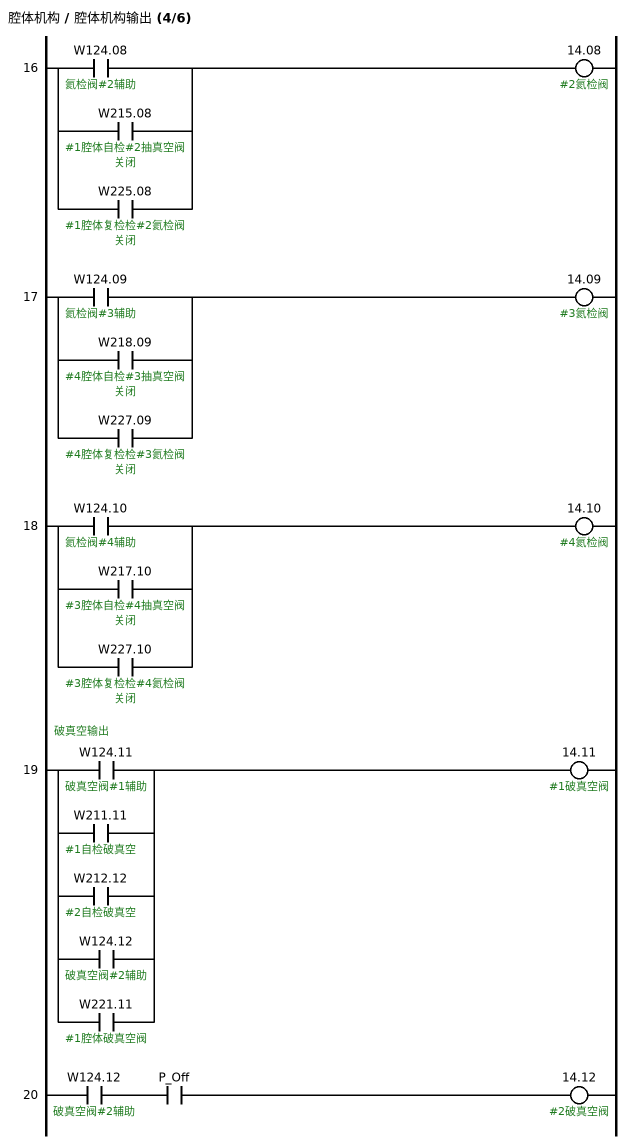
; rung 16
LD W124.08  ; 氦检阀#2辅助
OR W215.08  ; #1腔体自检#2抽真空阀关闭
OR W225.08  ; #1腔体复检检#2氦检阀关闭
OUT 14.08  ; #2氦检阀
; rung 17
LD W124.09  ; 氦检阀#3辅助
OR W218.09  ; #4腔体自检#3抽真空阀关闭
OR W227.09  ; #4腔体复检检#3氦检阀关闭
OUT 14.09  ; #3氦检阀
; rung 18
LD W124.10  ; 氦检阀#4辅助
OR W217.10  ; #3腔体自检#4抽真空阀关闭
OR W227.10  ; #3腔体复检检#4氦检阀关闭
OUT 14.10  ; #4氦检阀
; rung 19: 破真空输出
LD W124.11  ; 破真空阀#1辅助
OR W211.11  ; #1自检破真空
OR W212.12  ; #2自检破真空
OR W124.12  ; 破真空阀#2辅助
OR W221.11  ; #1腔体破真空阀
OUT 14.11  ; #1破真空阀
; rung 20
LD W124.12  ; 破真空阀#2辅助
AND P_Off
OUT 14.12  ; #2破真空阀

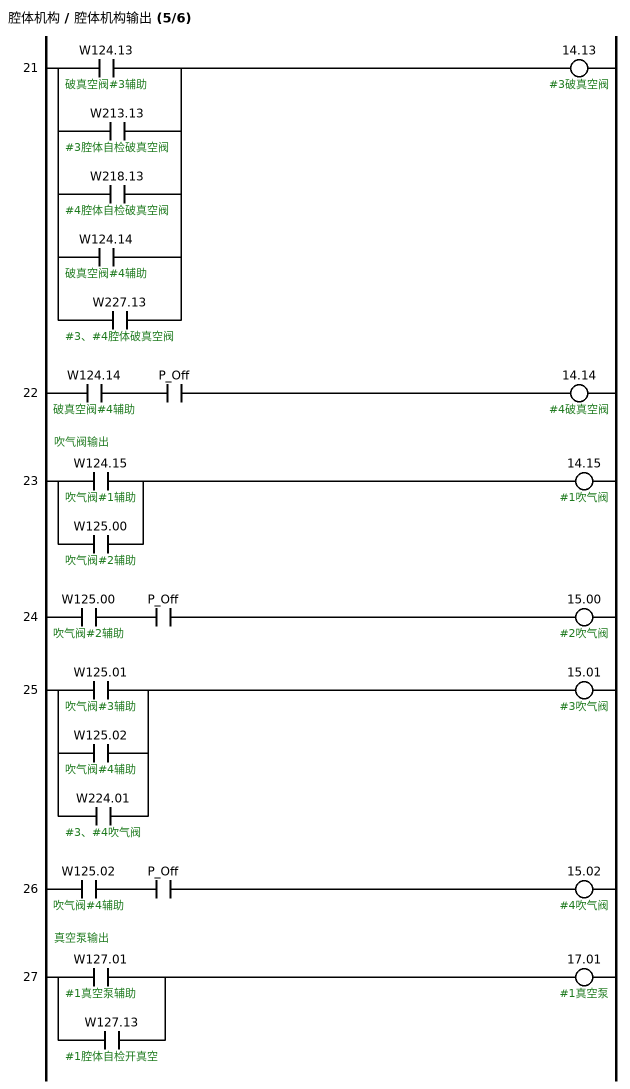
; rung 21
LD W124.13  ; 破真空阀#3辅助
OR W213.13  ; #3腔体自检破真空阀
OR W218.13  ; #4腔体自检破真空阀
OR W124.14  ; 破真空阀#4辅助
OR W227.13  ; #3、#4腔体破真空阀
OUT 14.13  ; #3破真空阀
; rung 22
LD W124.14  ; 破真空阀#4辅助
AND P_Off
OUT 14.14  ; #4破真空阀
; rung 23: 吹气阀输出
LD W124.15  ; 吹气阀#1辅助
OR W125.00  ; 吹气阀#2辅助
OUT 14.15  ; #1吹气阀
; rung 24
LD W125.00  ; 吹气阀#2辅助
AND P_Off
OUT 15.00  ; #2吹气阀
; rung 25
LD W125.01  ; 吹气阀#3辅助
OR W125.02  ; 吹气阀#4辅助
OR W224.01  ; #3、#4吹气阀
OUT 15.01  ; #3吹气阀
; rung 26
LD W125.02  ; 吹气阀#4辅助
AND P_Off
OUT 15.02  ; #4吹气阀
; rung 27: 真空泵输出
LD W127.01  ; #1真空泵辅助
OR W127.13  ; #1腔体自检开真空
OUT 17.01  ; #1真空泵

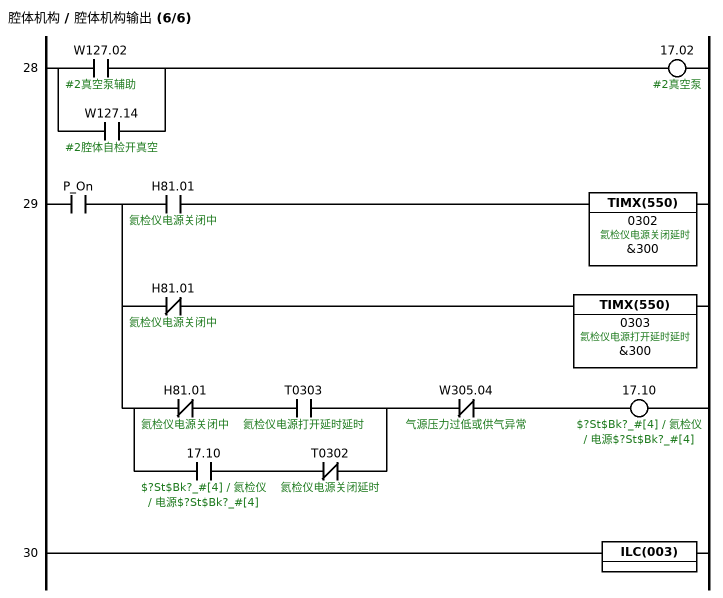
; rung 28
LD W127.02  ; #2真空泵辅助
OR W127.14  ; #2腔体自检开真空
OUT 17.02  ; #2真空泵
; rung 29
LD P_On
OUT TR0
AND H81.01  ; 氦检仪电源关闭中
TIMX(550) 0302 &300  ; 氦检仪电源关闭延时
LD TR0
ANDNOT H81.01  ; 氦检仪电源关闭中
TIMX(550) 0303 &300  ; 氦检仪电源打开延时延时
LD TR0
LDNOT H81.01  ; 氦检仪电源关闭中
AND T0303  ; 氦检仪电源打开延时延时
LD 17.10  ; $?St$Bk?_#[4] / 氦检仪 / 电源$?St$Bk?_#[4]
ANDNOT T0302  ; 氦检仪电源关闭延时
ORLD
ANDLD
ANDNOT W305.04  ; 气源压力过低或供气异常
OUT 17.10  ; $?St$Bk?_#[4] / 氦检仪 / 电源$?St$Bk?_#[4]
; rung 30
ILC(003)

### Section 工站复位

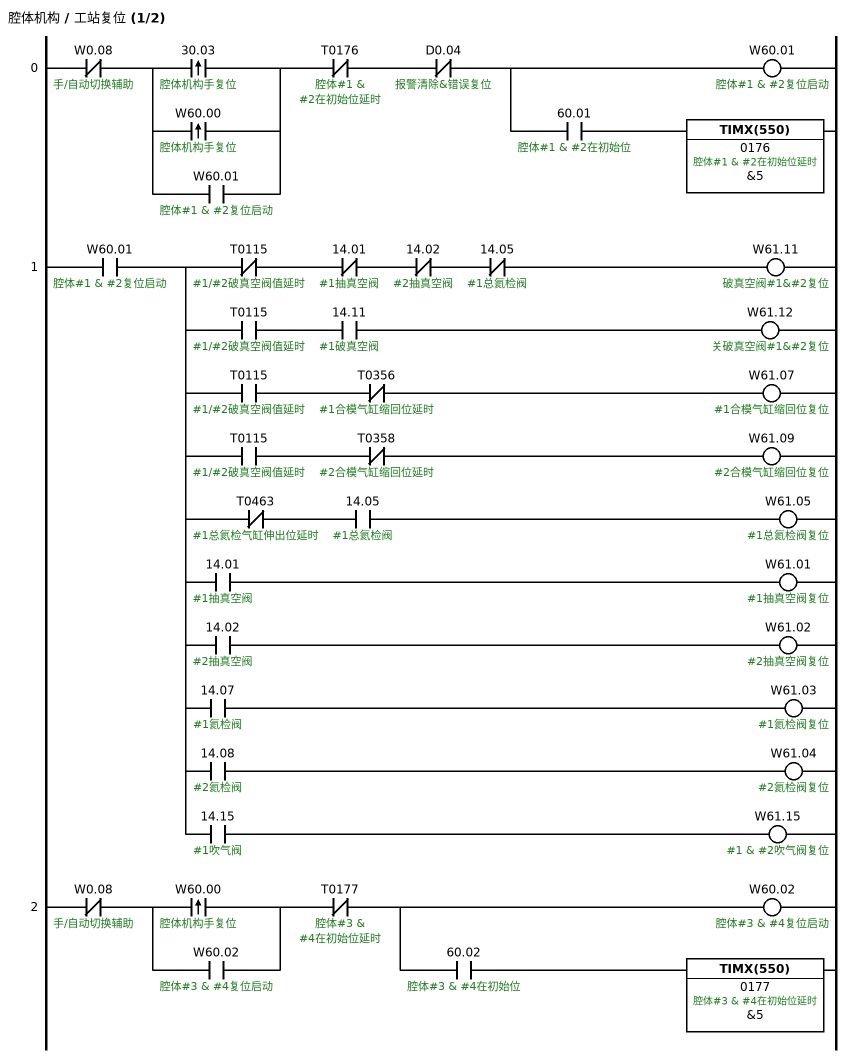
; rung 0
LDNOT W0.08  ; 手/自动切换辅助
@LD 30.03  ; 腔体机构手复位
@OR W60.00  ; 腔体机构手复位
OR W60.01  ; 腔体#1 & #2复位启动
ANDLD
ANDNOT T0176  ; 腔体#1 & #2在初始位延时
ANDNOT D0.04  ; 报警清除&错误复位
OUT W60.01  ; 腔体#1 & #2复位启动
AND 60.01  ; 腔体#1 & #2在初始位
TIMX(550) 0176 &5  ; 腔体#1 & #2在初始位延时
; rung 1
LD W60.01  ; 腔体#1 & #2复位启动
OUT TR0
ANDNOT T0115  ; #1/#2破真空阀值延时
ANDNOT 14.01  ; #1抽真空阀
ANDNOT 14.02  ; #2抽真空阀
ANDNOT 14.05  ; #1总氦检阀
OUT W61.11  ; 破真空阀#1&#2复位
LD TR0
AND T0115  ; #1/#2破真空阀值延时
AND 14.11  ; #1破真空阀
OUT W61.12  ; 关破真空阀#1&#2复位
LD TR0
AND T0115  ; #1/#2破真空阀值延时
ANDNOT T0356  ; #1合模气缸缩回位延时
OUT W61.07  ; #1合模气缸缩回位复位
LD TR0
AND T0115  ; #1/#2破真空阀值延时
ANDNOT T0358  ; #2合模气缸缩回位延时
OUT W61.09  ; #2合模气缸缩回位复位
LD TR0
ANDNOT T0463  ; #1总氦检气缸伸出位延时
AND 14.05  ; #1总氦检阀
OUT W61.05  ; #1总氦检阀复位
LD TR0
AND 14.01  ; #1抽真空阀
OUT W61.01  ; #1抽真空阀复位
LD TR0
AND 14.02  ; #2抽真空阀
OUT W61.02  ; #2抽真空阀复位
LD TR0
AND 14.07  ; #1氦检阀
OUT W61.03  ; #1氦检阀复位
LD TR0
AND 14.08  ; #2氦检阀
OUT W61.04  ; #2氦检阀复位
LD TR0
AND 14.15  ; #1吹气阀
OUT W61.15  ; #1 & #2吹气阀复位
; rung 2
LDNOT W0.08  ; 手/自动切换辅助
@LD W60.00  ; 腔体机构手复位
OR W60.02  ; 腔体#3 & #4复位启动
ANDLD
ANDNOT T0177  ; 腔体#3 & #4在初始位延时
OUT W60.02  ; 腔体#3 & #4复位启动
AND 60.02  ; 腔体#3 & #4在初始位
TIMX(550) 0177 &5  ; 腔体#3 & #4在初始位延时

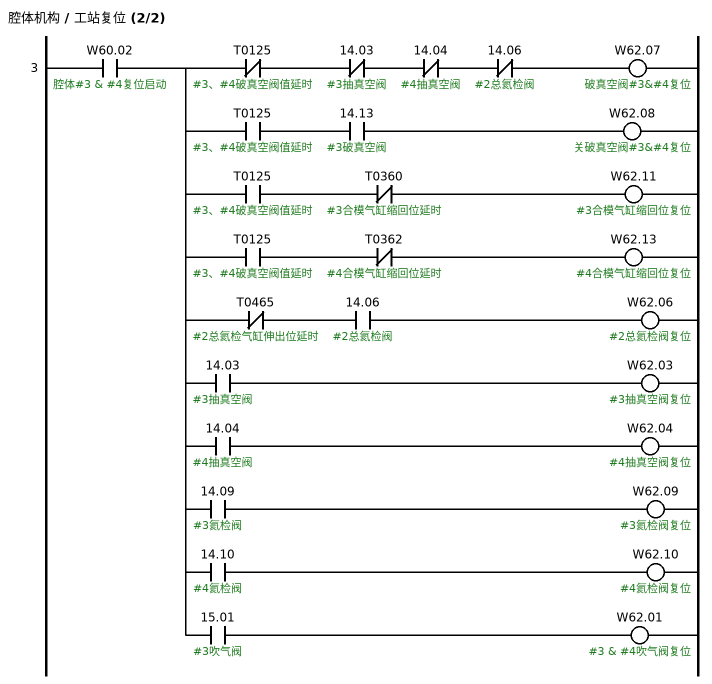
; rung 3
LD W60.02  ; 腔体#3 & #4复位启动
OUT TR0
ANDNOT T0125  ; #3、#4破真空阀值延时
ANDNOT 14.03  ; #3抽真空阀
ANDNOT 14.04  ; #4抽真空阀
ANDNOT 14.06  ; #2总氦检阀
OUT W62.07  ; 破真空阀#3&#4复位
LD TR0
AND T0125  ; #3、#4破真空阀值延时
AND 14.13  ; #3破真空阀
OUT W62.08  ; 关破真空阀#3&#4复位
LD TR0
AND T0125  ; #3、#4破真空阀值延时
ANDNOT T0360  ; #3合模气缸缩回位延时
OUT W62.11  ; #3合模气缸缩回位复位
LD TR0
AND T0125  ; #3、#4破真空阀值延时
ANDNOT T0362  ; #4合模气缸缩回位延时
OUT W62.13  ; #4合模气缸缩回位复位
LD TR0
ANDNOT T0465  ; #2总氦检气缸伸出位延时
AND 14.06  ; #2总氦检阀
OUT W62.06  ; #2总氦检阀复位
LD TR0
AND 14.03  ; #3抽真空阀
OUT W62.03  ; #3抽真空阀复位
LD TR0
AND 14.04  ; #4抽真空阀
OUT W62.04  ; #4抽真空阀复位
LD TR0
AND 14.09  ; #3氦检阀
OUT W62.09  ; #3氦检阀复位
LD TR0
AND 14.10  ; #4氦检阀
OUT W62.10  ; #4氦检阀复位
LD TR0
AND 15.01  ; #3吹气阀
OUT W62.01  ; #3 & #4吹气阀复位

### Section END
; rung 0
END(001)

## Program 出料机构 (cyclic task 4)

### Section 安全限制条件

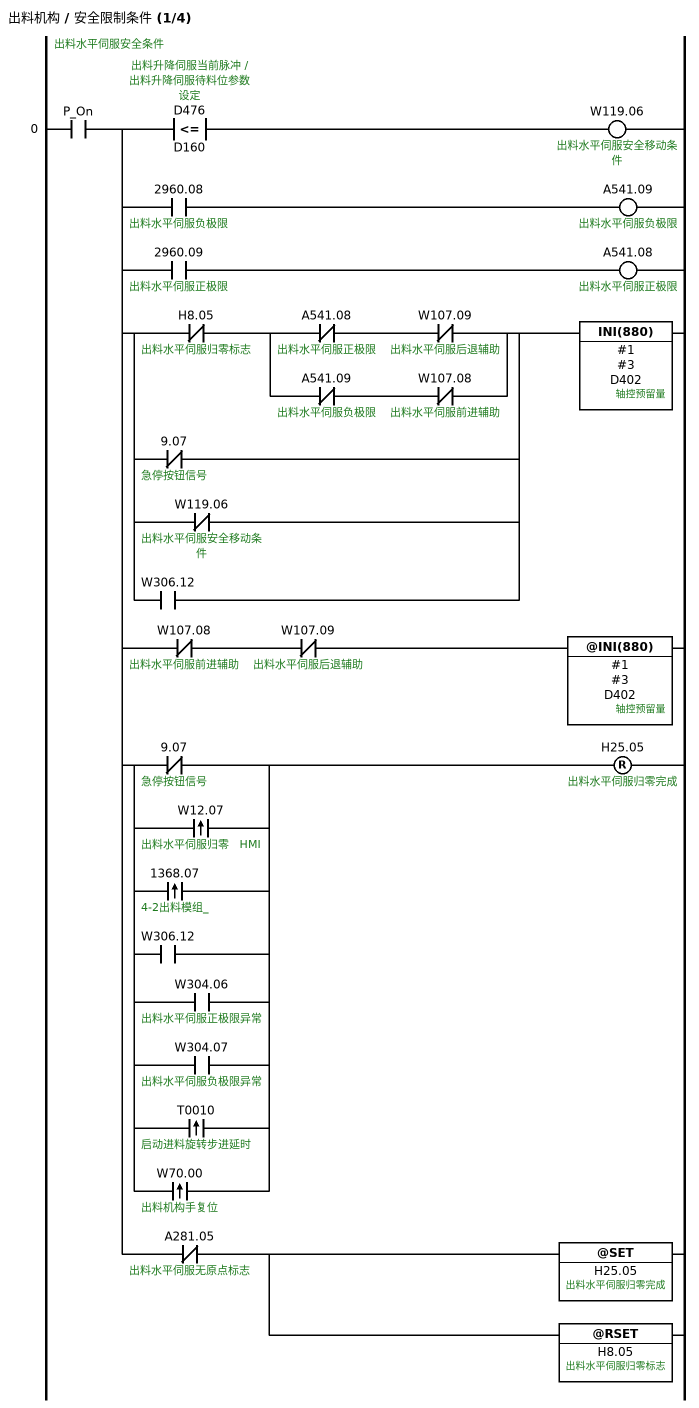
; rung 0: 出料水平伺服安全条件
LD P_On
OUT TR0
AND<=(315) D476 D160  ; 出料升降伺服当前脉冲, 出料升降伺服待料位参数设定
OUT W119.06  ; 出料水平伺服安全移动条件
LD TR0
AND 2960.08  ; 出料水平伺服负极限
OUT A541.09  ; 出料水平伺服负极限
LD TR0
AND 2960.09  ; 出料水平伺服正极限
OUT A541.08  ; 出料水平伺服正极限
LD TR0
LDNOT H8.05  ; 出料水平伺服归零标志
LDNOT A541.08  ; 出料水平伺服正极限
ANDNOT W107.09  ; 出料水平伺服后退辅助
LDNOT A541.09  ; 出料水平伺服负极限
ANDNOT W107.08  ; 出料水平伺服前进辅助
ORLD
ANDLD
ORNOT 9.07  ; 急停按钮信号
ORNOT W119.06  ; 出料水平伺服安全移动条件
OR W306.12
ANDLD
INI(880) #1 #3 D402  ; 轴控预留量
LD TR0
ANDNOT W107.08  ; 出料水平伺服前进辅助
ANDNOT W107.09  ; 出料水平伺服后退辅助
@INI(880) #1 #3 D402  ; 轴控预留量
LD TR0
LDNOT 9.07  ; 急停按钮信号
@OR W12.07  ; 出料水平伺服归零   HMI
@OR 1368.07  ; 4-2出料模组_
OR W306.12
OR W304.06  ; 出料水平伺服正极限异常
OR W304.07  ; 出料水平伺服负极限异常
@OR T0010  ; 启动进料旋转步进延时
@OR W70.00  ; 出料机构手复位
ANDLD
RSET H25.05  ; 出料水平伺服归零完成
LD TR0
ANDNOT A281.05  ; 出料水平伺服无原点标志
@SET H25.05  ; 出料水平伺服归零完成
@RSET H8.05  ; 出料水平伺服归零标志

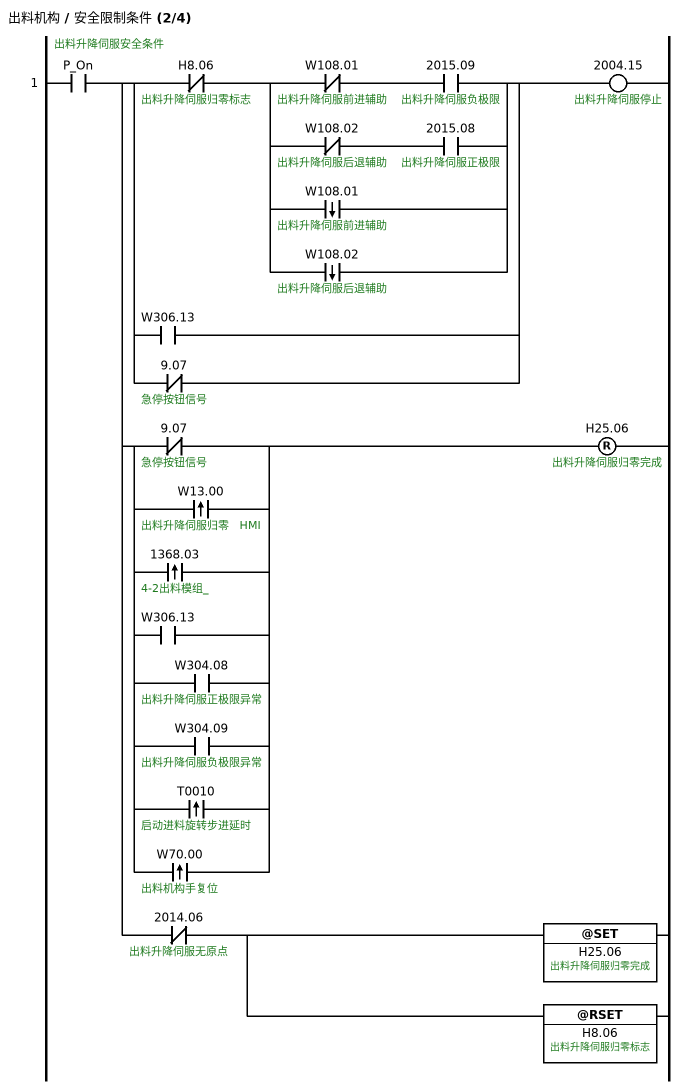
; rung 1: 出料升降伺服安全条件
LD P_On
OUT TR0
LDNOT H8.06  ; 出料升降伺服归零标志
LDNOT W108.01  ; 出料升降伺服前进辅助
AND 2015.09  ; 出料升降伺服负极限
LDNOT W108.02  ; 出料升降伺服后退辅助
AND 2015.08  ; 出料升降伺服正极限
ORLD
%OR W108.01  ; 出料升降伺服前进辅助
%OR W108.02  ; 出料升降伺服后退辅助
ANDLD
OR W306.13
ORNOT 9.07  ; 急停按钮信号
ANDLD
OUT 2004.15  ; 出料升降伺服停止
LD TR0
LDNOT 9.07  ; 急停按钮信号
@OR W13.00  ; 出料升降伺服归零   HMI
@OR 1368.03  ; 4-2出料模组_
OR W306.13
OR W304.08  ; 出料升降伺服正极限异常
OR W304.09  ; 出料升降伺服负极限异常
@OR T0010  ; 启动进料旋转步进延时
@OR W70.00  ; 出料机构手复位
ANDLD
RSET H25.06  ; 出料升降伺服归零完成
LD TR0
ANDNOT 2014.06  ; 出料升降伺服无原点
@SET H25.06  ; 出料升降伺服归零完成
@RSET H8.06  ; 出料升降伺服归零标志

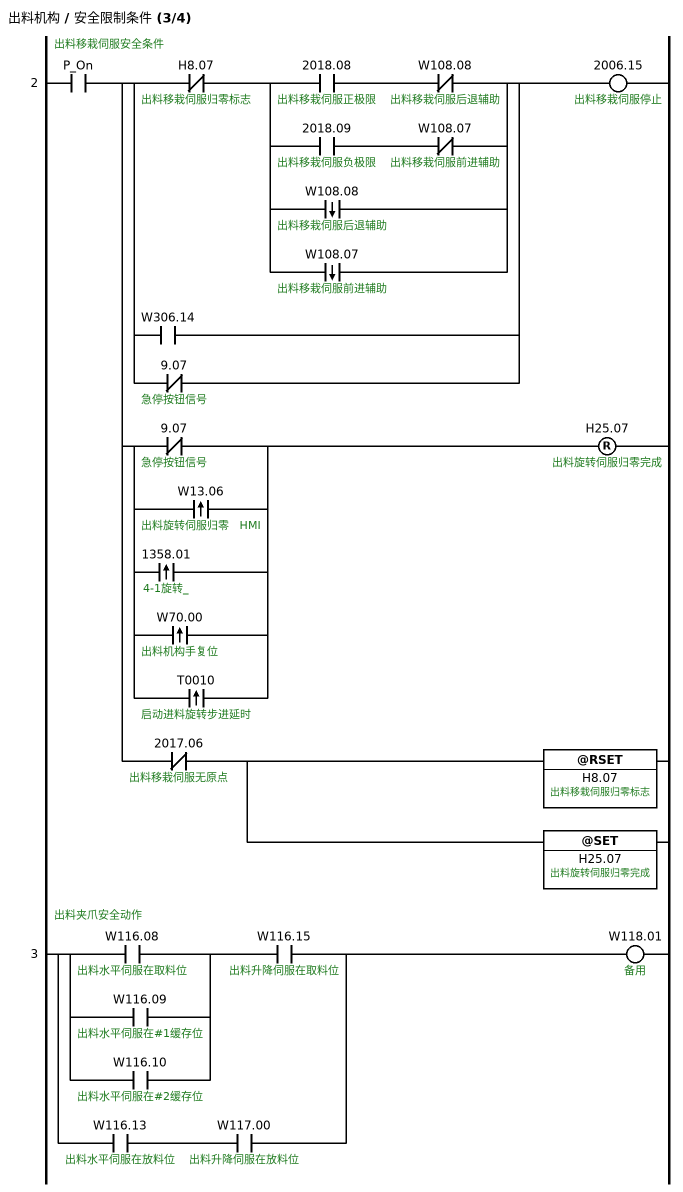
; rung 2: 出料移栽伺服安全条件
LD P_On
OUT TR0
LDNOT H8.07  ; 出料移栽伺服归零标志
LD 2018.08  ; 出料移栽伺服正极限
ANDNOT W108.08  ; 出料移栽伺服后退辅助
LD 2018.09  ; 出料移栽伺服负极限
ANDNOT W108.07  ; 出料移栽伺服前进辅助
ORLD
%OR W108.08  ; 出料移栽伺服后退辅助
%OR W108.07  ; 出料移栽伺服前进辅助
ANDLD
OR W306.14
ORNOT 9.07  ; 急停按钮信号
ANDLD
OUT 2006.15  ; 出料移栽伺服停止
LD TR0
LDNOT 9.07  ; 急停按钮信号
@OR W13.06  ; 出料旋转伺服归零   HMI
@OR 1358.01  ; 4-1旋转_
@OR W70.00  ; 出料机构手复位
@OR T0010  ; 启动进料旋转步进延时
ANDLD
RSET H25.07  ; 出料旋转伺服归零完成
LD TR0
ANDNOT 2017.06  ; 出料移栽伺服无原点
@RSET H8.07  ; 出料移栽伺服归零标志
@SET H25.07  ; 出料旋转伺服归零完成
; rung 3: 出料夹爪安全动作
LD W116.08  ; 出料水平伺服在取料位
OR W116.09  ; 出料水平伺服在#1缓存位
OR W116.10  ; 出料水平伺服在#2缓存位
AND W116.15  ; 出料升降伺服在取料位
LD W116.13  ; 出料水平伺服在放料位
AND W117.00  ; 出料升降伺服在放料位
ORLD
OUT W118.01  ; 备用

